TYPE TcaPushButtonConfig :
STRUCT
	LightState : eTcaPushButtonLightState;
	ButtonColor : eTcaPushButtonColor;
	ValidationTime	: TIME := T#100MS;
	FlashArray : ARRAY[0..128] OF TIME;
END_STRUCT
END_TYPE

(* stored: Version 1.1.0.1
   DUT TcaPushButtonConfig: Id {823b04db-e2d3-49ba-8c58-2830736d0faf} *)
